TYPE U_AXIS_INFO :
UNION

  stState             : ARRAY[1..MAX_AXIS] OF ST_AXIS_INFO;

  byState  AT %Q*     : ARRAY[1..MAX_AXIS] OF
                        ARRAY[1..SIZEOF(ST_AXIS_INFO)] OF BYTE;
END_UNION
END_TYPE

(* stored: Version 1.1.0.1, ProductVersion 3.1.4026.13
   DUT U_AXIS_INFO: Id {f1baede8-02ae-0ce0-0bf1-a621027ce175} *)
